LIN {X 0,Y 29.351,Z 476.14,A -85,B 0,C 180,E1 -30358.613,E2 -30358.613} C_VEL
LIN {X 0,Y 36.932,Z 474.38,A -85,B 0,C 180,E1 -30379.568,E2 -30379.568} C_VEL
LIN {X 0,Y 47.557,Z 471.456,A -85,B 0,C 180,E1 -30392.459,E2 -30392.459} C_VEL
LIN {X 0,Y 59.612,Z 467.297,A -85,B 0,C 180,E1 -30400.59,E2 -30400.59} C_VEL
LIN {X 0,Y 72.462,Z 461.794,A -85,B 0,C 180,E1 -30405.904,E2 -30405.904} C_VEL
LIN {X 0,Y 85.754,Z 454.797,A -85,B 0,C 180,E1 -30409.567,E2 -30409.567} C_VEL
LIN {X 0,Y 97.559,Z 447.315,A -85,B 0,C 180,E1 -30412.101,E2 -30412.101} C_VEL
LIN {X 0,Y 109.554,Z 438.293,A -85,B 0,C 180,E1 -30413.904,E2 -30413.904} C_VEL
LIN {X 0,Y 121.622,Z 427.442,A -85,B 0,C 180,E1 -30415.417,E2 -30415.417} C_VEL
LIN {X 0,Y 132.034,Z 416.273,A -85,B 0,C 180,E1 -30416.407,E2 -30416.407} C_VEL
LIN {X 0,Y 141.598,Z 404.023,A -85,B 0,C 180,E1 -30417.279,E2 -30417.279} C_VEL
LIN {X 0,Y 150.318,Z 390.543,A -85,B 0,C 180,E1 -30417.971,E2 -30417.971} C_VEL
LIN {X 0,Y 157.308,Z 377.288,A -85,B 0,C 180,E1 -30418.46,E2 -30418.46} C_VEL
LIN {X 0,Y 163.315,Z 363.08,A -85,B 0,C 180,E1 -30418.808,E2 -30418.808} C_VEL
LIN {X 0,Y 168.117,Z 348.171,A -85,B 0,C 180,E1 -30419.054,E2 -30419.054} C_VEL
LIN {X 0,Y 171.319,Z 334.167,A -85,B 0,C 180,E1 -30419.303,E2 -30419.303} C_VEL
LIN {X 0,Y 171.381,Z 333.752,A -85,B 0,C 180,E1 -30420,E2 -30420} C_VEL
LIN {X 0,Y 171.309,Z 334.21,A -85,B 0,C 180,E1 -30420.91,E2 -30420.91} C_VEL
LIN {X 0,Y 168.048,Z 348.377,A -85,B 0,C 180,E1 -30421.109,E2 -30421.109} C_VEL
LIN {X 0,Y 167.969,Z 348.938,A -85,B 0,C 180,E1 -30421.114,E2 -30421.114} C_VEL
LIN {X 0,Y 167.969,Z 416.971,A -85,B 0,C 180,E1 -30421.114,E2 -30421.114} C_VEL
LIN {X 0,Y 146.091,Z 416.971,A -85,B 0,C 180,E1 -30420.172,E2 -30420.172} C_VEL
LIN {X 0,Y 144.107,Z 414.971,A -85,B 0,C 180,E1 -30420.073,E2 -30420.073} C_VEL
LIN {X 0,Y 144.107,Z 406.332,A -85,B 0,C 180,E1 -30420.073,E2 -30420.073} C_VEL
LIN {X 0,Y 140.562,Z 405.122,A -85,B 0,C 180,E1 -30420.307,E2 -30420.307} C_VEL
LIN {X 0,Y 131.791,Z 416.172,A -85,B 0,C 180,E1 -30420.881,E2 -30420.881} C_VEL
LIN {X 0,Y 121.286,Z 427.313,A -85,B 0,C 180,E1 -30421.692,E2 -30421.692} C_VEL
LIN {X 0,Y 109.069,Z 438.128,A -85,B 0,C 180,E1 -30422.85,E2 -30422.85} C_VEL
LIN {X 0,Y 96.815,Z 447.178,A -85,B 0,C 180,E1 -30424.332,E2 -30424.332} C_VEL
LIN {X 0,Y 84.856,Z 454.559,A -85,B 0,C 180,E1 -30426.348,E2 -30426.348} C_VEL
LIN {X 0,Y 74.588,Z 459.909,A -85,B 0,C 180,E1 -30428.368,E2 -30428.368} C_VEL
LIN {X 0,Y 61.123,Z 465.746,A -85,B 0,C 180,E1 -30432.221,E2 -30432.221} C_VEL
LIN {X 0,Y 51.26,Z 469.203,A -85,B 0,C 180,E1 -30436.315,E2 -30436.315} C_VEL
LIN {X 0,Y 38.775,Z 472.696,A -85,B 0,C 180,E1 -30445.009,E2 -30445.009} C_VEL
LIN {X 0,Y 27.83,Z 474.999,A -85,B 0,C 180,E1 -30460.748,E2 -30460.748} C_VEL
LIN {X 0,Y 20.77,Z 476.164,A -85,B 0,C 180,E1 -30490.224,E2 -30490.224} C_VEL
LIN {X 0,Y 19.973,Z 476.317,A -85,B 0,C 180,E1 -30510.001,E2 -30510.001} C_VEL
LIN {X 0,Y 23.559,Z 475.748,A -85,B 0,C 180,E1 -30546.631,E2 -30546.631} C_VEL
LIN {X 0,Y 32.962,Z 474.055,A -85,B 0,C 180,E1 -30568.524,E2 -30568.524} C_VEL
LIN {X 0,Y 44.903,Z 471.195,A -85,B 0,C 180,E1 -30579.9,E2 -30579.9} C_VEL
LIN {X 0,Y 57.799,Z 467.103,A -85,B 0,C 180,E1 -30586.595,E2 -30586.595} C_VEL
LIN {X 0,Y 71.18,Z 461.678,A -85,B 0,C 180,E1 -30590.879,E2 -30590.879} C_VEL
LIN {X 0,Y 81.407,Z 456.618,A -85,B 0,C 180,E1 -30593.128,E2 -30593.128} C_VEL
LIN {X 0,Y 91.723,Z 450.686,A -85,B 0,C 180,E1 -30594.93,E2 -30594.93} C_VEL
LIN {X 0,Y 103.841,Z 442.444,A -85,B 0,C 180,E1 -30596.653,E2 -30596.653} C_VEL
LIN {X 0,Y 116.039,Z 432.512,A -85,B 0,C 180,E1 -30597.92,E2 -30597.92} C_VEL
LIN {X 0,Y 126.531,Z 422.336,A -85,B 0,C 180,E1 -30598.825,E2 -30598.825} C_VEL
LIN {X 0,Y 137.051,Z 410.212,A -85,B 0,C 180,E1 -30599.555,E2 -30599.555} C_VEL
LIN {X 0,Y 140.561,Z 405.572,A -85,B 0,C 180,E1 -30599.804,E2 -30599.804} C_VEL
LIN {X 0,Y 140.561,Z 405.574,A -85,B 0,C 180,E1 -30599.888,E2 -30599.888} C_VEL
LIN {X 0,Y 131.781,Z 416.577,A -85,B 0,C 180,E1 -30600.513,E2 -30600.513} C_VEL
LIN {X 0,Y 121.262,Z 427.696,A -85,B 0,C 180,E1 -30601.25,E2 -30601.25} C_VEL
LIN {X 0,Y 109.025,Z 438.483,A -85,B 0,C 180,E1 -30602.333,E2 -30602.333} C_VEL
LIN {X 0,Y 96.673,Z 447.581,A -85,B 0,C 180,E1 -30603.804,E2 -30603.804} C_VEL
LIN {X 0,Y 84.754,Z 454.928,A -85,B 0,C 180,E1 -30605.689,E2 -30605.689} C_VEL
LIN {X 0,Y 71.059,Z 461.878,A -85,B 0,C 180,E1 -30608.491,E2 -30608.491} C_VEL
LIN {X 0,Y 57.636,Z 467.343,A -85,B 0,C 180,E1 -30612.706,E2 -30612.706} C_VEL
LIN {X 0,Y 44.715,Z 471.475,A -85,B 0,C 180,E1 -30619.43,E2 -30619.43} C_VEL
LIN {X 0,Y 32.766,Z 474.371,A -85,B 0,C 180,E1 -30630.911,E2 -30630.911} C_VEL
LIN {X 0,Y 23.337,Z 476.098,A -85,B 0,C 180,E1 -30652.963,E2 -30652.963} C_VEL
LIN {X 0,Y 19.88,Z 476.69,A -85,B 0,C 180,E1 -30689.999,E2 -30689.999} C_VEL
LIN {X 0,Y 23.334,Z 476.073,A -85,B 0,C 180,E1 -30727.04,E2 -30727.04} C_VEL
LIN {X 0,Y 32.756,Z 474.313,A -85,B 0,C 180,E1 -30749.116,E2 -30749.116} C_VEL
LIN {X 0,Y 44.693,Z 471.388,A -85,B 0,C 180,E1 -30760.648,E2 -30760.648} C_VEL
LIN {X 0,Y 57.63,Z 467.229,A -85,B 0,C 180,E1 -30767.317,E2 -30767.317} C_VEL
LIN {X 0,Y 71.058,Z 461.726,A -85,B 0,C 180,E1 -30771.513,E2 -30771.513} C_VEL
LIN {X 0,Y 81.316,Z 456.611,A -85,B 0,C 180,E1 -30773.68,E2 -30773.68} C_VEL
LIN {X 0,Y 93.367,Z 449.486,A -85,B 0,C 180,E1 -30775.838,E2 -30775.838} C_VEL
LIN {X 0,Y 105.538,Z 440.934,A -85,B 0,C 180,E1 -30777.284,E2 -30777.284} C_VEL
LIN {X 0,Y 117.759,Z 430.64,A -85,B 0,C 180,E1 -30778.497,E2 -30778.497} C_VEL
LIN {X 0,Y 128.271,Z 420.108,A -85,B 0,C 180,E1 -30779.272,E2 -30779.272} C_VEL
LIN {X 0,Y 137.925,Z 408.65,A -85,B 0,C 180,E1 -30779.94,E2 -30779.94} C_VEL
LIN {X 0,Y 140.56,Z 405.127,A -85,B 0,C 180,E1 -30780.105,E2 -30780.105} C_VEL
LIN {X 0,Y 140.562,Z 405.122,A -85,B 0,C 180,E1 -30780.307,E2 -30780.307} C_VEL
LIN {X 0,Y 140.587,Z 407.122,A -85,B 0,C 180,E1 -30781.13,E2 -30781.13} C_VEL
LIN {X 0,Y 140.587,Z 460.435,A -85,B 0,C 180,E1 -30781.13,E2 -30781.13} C_VEL
LIN {X 0,Y 96.34,Z 460.435,A -85,B 0,C 180,E1 -30780.387,E2 -30780.387} C_VEL
LIN {X 0,Y 94.342,Z 458.435,A -85,B 0,C 180,E1 -30780.337,E2 -30780.337} C_VEL
LIN {X 0,Y 94.342,Z 452.243,A -85,B 0,C 180,E1 -30780.337,E2 -30780.337} C_VEL
LIN {X 0,Y 91.371,Z 450.526,A -85,B 0,C 180,E1 -30780.691,E2 -30780.691} C_VEL
LIN {X 0,Y 80.867,Z 456.5,A -85,B 0,C 180,E1 -30781.908,E2 -30781.908} C_VEL
LIN {X 0,Y 66.937,Z 463.075,A -85,B 0,C 180,E1 -30784.096,E2 -30784.096} C_VEL
LIN {X 0,Y 56.573,Z 467.05,A -85,B 0,C 180,E1 -30786.365,E2 -30786.365} C_VEL
LIN {X 0,Y 42.971,Z 471.17,A -85,B 0,C 180,E1 -30791.096,E2 -30791.096} C_VEL
LIN {X 0,Y 29.873,Z 474.06,A -85,B 0,C 180,E1 -30799.773,E2 -30799.773} C_VEL
LIN {X 0,Y 18.349,Z 475.788,A -85,B 0,C 180,E1 -30820.003,E2 -30820.003} C_VEL
LIN {X 0,Y 12.87,Z 476.384,A -85,B 0,C 180,E1 -30870.001,E2 -30870.001} C_VEL
LIN {X 0,Y 18.338,Z 475.815,A -85,B 0,C 180,E1 -30920.041,E2 -30920.041} C_VEL
LIN {X 0,Y 29.862,Z 474.121,A -85,B 0,C 180,E1 -30940.29,E2 -30940.29} C_VEL
LIN {X 0,Y 42.974,Z 471.261,A -85,B 0,C 180,E1 -30948.889,E2 -30948.889} C_VEL
LIN {X 0,Y 56.572,Z 467.169,A -85,B 0,C 180,E1 -30953.65,E2 -30953.65} C_VEL
LIN {X 0,Y 70.402,Z 461.744,A -85,B 0,C 180,E1 -30956.635,E2 -30956.635} C_VEL
LIN {X 0,Y 80.865,Z 456.683,A -85,B 0,C 180,E1 -30958.15,E2 -30958.15} C_VEL
LIN {X 0,Y 91.369,Z 450.751,A -85,B 0,C 180,E1 -30959.425,E2 -30959.425} C_VEL
LIN {X 0,Y 91.542,Z 450.647,A -85,B 0,C 180,E1 -30960,E2 -30960} C_VEL
LIN {X 0,Y 77.345,Z 458.536,A -85,B 0,C 180,E1 -30961.752,E2 -30961.752} C_VEL
LIN {X 0,Y 63.406,Z 464.719,A -85,B 0,C 180,E1 -30963.993,E2 -30963.993} C_VEL
LIN {X 0,Y 49.641,Z 469.502,A -85,B 0,C 180,E1 -30967.677,E2 -30967.677} C_VEL
LIN {X 0,Y 36.202,Z 473.006,A -85,B 0,C 180,E1 -30973.909,E2 -30973.909} C_VEL
LIN {X 0,Y 23.582,Z 475.31,A -85,B 0,C 180,E1 -30986.607,E2 -30986.607} C_VEL
LIN {X 0,Y 14.095,Z 476.469,A -85,B 0,C 180,E1 -31020.09,E2 -31020.09} C_VEL
LIN {X 0,Y 12.767,Z 476.623,A -85,B 0,C 180,E1 -31049.999,E2 -31049.999} C_VEL
LIN {X 0,Y 18.14,Z 476.006,A -85,B 0,C 180,E1 -31100.793,E2 -31100.793} C_VEL
LIN {X 0,Y 29.721,Z 474.246,A -85,B 0,C 180,E1 -31121.057,E2 -31121.057} C_VEL
LIN {X 0,Y 42.854,Z 471.321,A -85,B 0,C 180,E1 -31129.735,E2 -31129.735} C_VEL
LIN {X 0,Y 56.491,Z 467.161,A -85,B 0,C 180,E1 -31134.428,E2 -31134.428} C_VEL
LIN {X 0,Y 70.359,Z 461.658,A -85,B 0,C 180,E1 -31137.29,E2 -31137.29} C_VEL
LIN {X 0,Y 80.841,Z 456.543,A -85,B 0,C 180,E1 -31138.743,E2 -31138.743} C_VEL
LIN {X 0,Y 91.364,Z 450.536,A -85,B 0,C 180,E1 -31140.075,E2 -31140.075} C_VEL
LIN {X 0,Y 91.371,Z 450.526,A -85,B 0,C 180,E1 -31140.691,E2 -31140.691} C_VEL
LIN {X 0,Y 91.417,Z 452.526,A -85,B 0,C 180,E1 -31141.956,E2 -31141.956} C_VEL
LIN {X 0,Y 91.417,Z 480.25,A -85,B 0,C 180,E1 -31141.956,E2 -31141.956} C_VEL
LIN {X 0,Y 49.379,Z 480.25,A -85,B 0,C 180,E1 -31139.197,E2 -31139.197} C_VEL
LIN {X 0,Y 47.391,Z 478.25,A -85,B 0,C 180,E1 -31138.945,E2 -31138.945} C_VEL
LIN {X 0,Y 47.391,Z 472.454,A -85,B 0,C 180,E1 -31138.945,E2 -31138.945} C_VEL
LIN {X 0,Y 45.088,Z 470.507,A -85,B 0,C 180,E1 -31140.001,E2 -31140.001} C_VEL
LIN {X 0,Y 42.182,Z 471.238,A -85,B 0,C 180,E1 -31141.511,E2 -31141.511} C_VEL
LIN {X 0,Y 28.268,Z 474.127,A -85,B 0,C 180,E1 -31146.027,E2 -31146.027} C_VEL
LIN {X 0,Y 14.814,Z 475.855,A -85,B 0,C 180,E1 -31158.406,E2 -31158.406} C_VEL
LIN {X 0,Y 5.759,Z 476.45,A -85,B 0,C 180,E1 -31230.003,E2 -31230.003} C_VEL
LIN {X 0,Y 14.808,Z 475.881,A -85,B 0,C 180,E1 -31301.665,E2 -31301.665} C_VEL
LIN {X 0,Y 28.265,Z 474.187,A -85,B 0,C 180,E1 -31314.034,E2 -31314.034} C_VEL
LIN {X 0,Y 42.184,Z 471.327,A -85,B 0,C 180,E1 -31318.46,E2 -31318.46} C_VEL
LIN {X 0,Y 45.805,Z 470.412,A -85,B 0,C 180,E1 -31319.999,E2 -31319.999} C_VEL
LIN {X 0,Y 35.174,Z 472.94,A -85,B 0,C 180,E1 -31322.505,E2 -31322.505} C_VEL
LIN {X 0,Y 21.358,Z 475.244,A -85,B 0,C 180,E1 -31329.175,E2 -31329.175} C_VEL
LIN {X 0,Y 8.677,Z 476.403,A -85,B 0,C 180,E1 -31355.908,E2 -31355.908} C_VEL
LIN {X 0,Y 5.665,Z 476.557,A -85,B 0,C 180,E1 -31409.997,E2 -31409.997} C_VEL
LIN {X 0,Y 14.704,Z 475.939,A -85,B 0,C 180,E1 -31482.92,E2 -31482.92} C_VEL
LIN {X 0,Y 28.222,Z 474.178,A -85,B 0,C 180,E1 -31494.941,E2 -31494.941} C_VEL
LIN {X 0,Y 42.17,Z 471.253,A -85,B 0,C 180,E1 -31499.387,E2 -31499.387} C_VEL
LIN {X 0,Y 45.088,Z 470.507,A -85,B 0,C 180,E1 -31500.001,E2 -31500.001} C_VEL
LIN {X 0,Y 47.549,Z 472.446,A -85,B 0,C 180,E1 -31500.46,E2 -31500.46} C_VEL
LIN {X 0,Y 47.549,Z 600,A -85,B 0,C 180,E1 -31500.46,E2 -31500.46} C_VEL
LIN {X 0,Y 47.549,Z 600,A -85,B 0,C 180,E1 -31500.46,E2 -31500.46}

QRS_NEXT_CUT()

QRS_NEXT()
QRS_HOME()

END
